KUKA KRL program: UP202.src, UP202.dat

--- UP202.src ---
&ACCESS RV1
&COMMENT WERKZEUGWECHSEL G1
&PARAM EDITMASK = Up999[1-999]
&PARAM TEMPLATE = C:\KRC\Roboter\Template\upvorgabe
&PARAM TPVW_VERSION = 8.3.18
&PARAM DISKPATH = UPs
DEF UP202()
; FOLD UP Anfang;%{SE} %MKUKATPVW
SPS_N=-1
SPS_FERTIG=FALSE
IF NOT CALLBYSELECT THEN
INTERRUPT DECL 10 WHEN $CYCFLAG[254]==FALSE DO VW(#FB_STOP,TRUE)
INTERRUPT ON 10
INT10=TRUE
VW_USR_R (#USR_INIT)
ENDIF
VW(#VW_INIT_UP,TRUE)
; ENDFOLD
;FOLD -- ********************************************** -- ;%{PSE}%MKUKATPVW,%CVW_COM,%VCOMMENT,%P 1:Comment:, 2:**********************************************
;FOLD {H}
M_COMMENT("**********************************************")
;ENDFOLD
;ENDFOLD
;FOLD -- Modell :  VW316/7 -- ;%{PSE}%MKUKATPVW,%CVW_COM,%VCOMMENT,%P 1:Comment:, 2:Modell :  VW316/7
;FOLD {H}
M_COMMENT("Modell :  VW316/7")
;ENDFOLD
;ENDFOLD
;FOLD -- Line   :  TVOL -- ;%{PSE}%MKUKATPVW,%CVW_COM,%VCOMMENT,%P 1:Comment:, 2:Line   :  TVOL
;FOLD {H}
M_COMMENT("Line   :  TVOL")
;ENDFOLD
;ENDFOLD
;FOLD -- Robot  :  5100R01 -- ;%{PSE}%MKUKATPVW,%CVW_COM,%VCOMMENT,%P 1:Comment:, 2:Robot  :  5100R01
;FOLD {H}
M_COMMENT("Robot  :  5100R01")
;ENDFOLD
;ENDFOLD
;FOLD -- Arbeit :  WERKZEUGWECHSEL G2 -- ;%{PSE}%MKUKATPVW,%CVW_COM,%VCOMMENT,%P 1:Comment:, 2:Arbeit :  WERKZEUGWECHSEL G2
;FOLD {H}
M_COMMENT("Arbeit :  WERKZEUGWECHSEL G2")
;ENDFOLD
;ENDFOLD
;FOLD -- ********************************************** -- ;%{PSE}%MKUKATPVW,%CVW_COM,%VCOMMENT,%P 1:Comment:, 2:**********************************************
;FOLD {H}
M_COMMENT("**********************************************")
;ENDFOLD
;ENDFOLD
;FOLD PTP VB=100% VE=0% ACC=100% RobWzg=2 Base=0 SPSTrig=5[1/100s] P;%{P}%MKUKATPVW,%CMOVE8,%VPTP,%P 1:1, 2: VB=, 3:100, 4:%, 5: VE=, 6:0, 7:%, 8: ACC=, 9:100, 10:%, 11: RobWzg=, 12:2, 13: Base=, 14:0, 15: SPSTrig=, 16:5, 17:[1/100s], 18: P, 19:1, 20:-1, 21:1
;FOLD 1:  FB PSPS = EIN;%{SE}%MKUKATPVW %CVW_SPS %VFBPSPS %P 2:FB PSPS = EIN,3:   FBPSPS
;ENDFOLD
;FOLD 2:  -- Initialisierung Merker --;%{SE}%MKUKATPVW %CVW_COM %VCOMMENT %P 2: -- Initialisierung Merker --,3:  VW_COMMENT
;ENDFOLD
;FOLD 3:  SPSMAKRO50 = EIN;%{SE}%MKUKATPVW %CVW_SPS %VMAKRO %P 2:SPSMAKRO50 = EIN,3:   MAKRO
;ENDFOLD
;FOLD 4:  SPSMAKRO51 = EIN;%{SE}%MKUKATPVW %CVW_SPS %VMAKRO %P 2:SPSMAKRO51 = EIN,3:   MAKRO
;ENDFOLD
;FOLD 5:  -- Profilfrei --;%{SE}%MKUKATPVW %CVW_COM %VCOMMENT %P 2: -- Profilfrei --,3:  VW_COMMENT
;ENDFOLD
;FOLD 6:  SPSMAKRO46 = EIN;%{SE}%MKUKATPVW %CVW_SPS %VMAKRO %P 2:SPSMAKRO46 = EIN,3:   MAKRO
;ENDFOLD
;FOLD 7:  -- Verriegelungen Freigabe --;%{SE}%MKUKATPVW %CVW_COM %VCOMMENT %P 2: -- Verriegelungen Freigabe --,3:  VW_COMMENT
;ENDFOLD
;FOLD 8:  SPSMAKRO45 = EIN;%{SE}%MKUKATPVW %CVW_SPS %VMAKRO %P 2:SPSMAKRO45 = EIN,3:   MAKRO
;ENDFOLD
;FOLD 9:  -- Greifer Initialisieren --;%{SE}%MKUKATPVW %CVW_COM %VCOMMENT %P 2: -- Greifer Initialisieren --,3:  VW_COMMENT
;ENDFOLD
;FOLD 10:  F1 = EIN;%{SE}%MKUKATPVW %CVW_SPS %VBOASG %P 2:F1 = EIN,3:   BOASG
;ENDFOLD
;FOLD 11:  F2 = EIN;%{SE}%MKUKATPVW %CVW_SPS %VBOASG %P 2:F2 = EIN,3:   BOASG
;ENDFOLD
;FOLD 12:  F3 = EIN;%{SE}%MKUKATPVW %CVW_SPS %VBOASG %P 2:F3 = EIN,3:   BOASG
;ENDFOLD
;FOLD 13:  F17 = EIN;%{SE}%MKUKATPVW %CVW_SPS %VBOASG %P 2:F17 = EIN,3:   BOASG
;ENDFOLD
;FOLD 14:  M190 = E605 + E603;%{SE}%MKUKATPVW %CVW_SPS %VBOASG %P 2:M190 = E605 + E603,3:   BOASG
;ENDFOLD
;FOLD 15:  SPSMAKRO342 = EIN;%{SE}%MKUKATPVW %CVW_SPS %VMAKRO %P 2:SPSMAKRO342 = EIN,3:   MAKRO
;ENDFOLD
;FOLD 16:  SPSMAKRO340 = EIN;%{SE}%MKUKATPVW %CVW_SPS %VMAKRO %P 2:SPSMAKRO340 = EIN,3:   MAKRO
;ENDFOLD
;FOLD 17:  WARTE BIS M31 & M33 & M35 & M1;%{SE}%MKUKATPVW %CVW_SPS %VWBOASG %P 2:WARTE BIS M31 & M33 & M35 & M1,3:   WBOASG
;ENDFOLD
;FOLD 18:  WARTE BIS E23;%{SE}%MKUKATPVW %CVW_SPS %VWBOASG %P 2:WARTE BIS E23,3:   WBOASG
;ENDFOLD
;FOLD 19:  FB PSPS = M30 & M1 & M31 & M33 & M35;%{SE}%MKUKATPVW %CVW_SPS %VFBPSPS %P 2:FB PSPS = M30 & M1 & M31 & M33 & M35,3:   FBPSPS
;ENDFOLD
;FOLD {H}
VW_MPARA_ACT=P1_D
Act_P1 = P1
Act_P2 = P1
VW(#MPARA,TRUE)
SPS_FERTIG=FALSE
TRIGGER WHEN DISTANCE=1 DELAY=-50 DO SPS_TRIG(1) PRIO=-1
PTP P1
$ADVANCE=1
WAIT FOR SPS_FERTIG
;ENDFOLD
;ENDFOLD
;FOLD -- Werkzeugwechselposition -- ;%{PSE}%MKUKATPVW,%CVW_COM,%VCOMMENT,%P 1:Comment:, 2:Werkzeugwechselposition
;FOLD {H}
M_COMMENT("Werkzeugwechselposition")
;ENDFOLD
;ENDFOLD
;FOLD PTP VB=100% VE=0% ACC=100% RobWzg=2 Base=0 SPSTrig=5[1/100s] P;%{P}%MKUKATPVW,%CMOVE8,%VPTP,%P 1:1, 2: VB=, 3:100, 4:%, 5: VE=, 6:0, 7:%, 8: ACC=, 9:100, 10:%, 11: RobWzg=, 12:2, 13: Base=, 14:0, 15: SPSTrig=, 16:5, 17:[1/100s], 18: P, 19:2, 20:-1, 21:2
;FOLD 1:  FB PSPS = EIN;%{SE}%MKUKATPVW %CVW_SPS %VFBPSPS %P 2:FB PSPS = EIN,3:   FBPSPS
;ENDFOLD
;FOLD 2:  -- Roboter ist in Wartungsstellung --;%{SE}%MKUKATPVW %CVW_COM %VCOMMENT %P 2: -- Roboter ist in Wartungsstellung --,3:  VW_COMMENT
;ENDFOLD
;FOLD 3:  A17 = EIN;%{SE}%MKUKATPVW %CVW_SPS %VBOASG %P 2:A17 = EIN,3:   BOASG
;ENDFOLD
;FOLD 4:  -- Prozessgeraet BMS --;%{SE}%MKUKATPVW %CVW_COM %VCOMMENT %P 2: -- Prozessgeraet BMS --,3:  VW_COMMENT
;ENDFOLD
;FOLD 5:  TECH4 Prozessgeraet  Handling    Greifer=Nr2  in Wartungsstellung   Techaufruf= EIN ;%{SE}%MKUKATPVW %CVW_SPS %VUSER %P 2:    TECH4.Prozessgeraet CN=403 P1=1 P2=0 P3=12 P4=20 P5=0 P6=0 P7=0 P8=0 P9=0 P10=EIN,3:   USER
;ENDFOLD
;FOLD 6:  -- Warte Wartungsstellung Ende --;%{SE}%MKUKATPVW %CVW_COM %VCOMMENT %P 2: -- Warte Wartungsstellung Ende --,3:  VW_COMMENT
;ENDFOLD
;FOLD 7:  WARTE BIS E17;%{SE}%MKUKATPVW %CVW_SPS %VWBOASG %P 2:WARTE BIS E17,3:   WBOASG
;ENDFOLD
;FOLD 8:  -- Wartungsstellung Ende --;%{SE}%MKUKATPVW %CVW_COM %VCOMMENT %P 2: -- Wartungsstellung Ende --,3:  VW_COMMENT
;ENDFOLD
;FOLD 9:  A17 = AUS;%{SE}%MKUKATPVW %CVW_SPS %VBOASG %P 2:A17 = AUS,3:   BOASG
;ENDFOLD
;FOLD 10:  WARTE BIS E23;%{SE}%MKUKATPVW %CVW_SPS %VWBOASG %P 2:WARTE BIS E23,3:   WBOASG
;ENDFOLD
;FOLD 11:  FB PSPS = M30 & M1 & M31 & M33 & M35;%{SE}%MKUKATPVW %CVW_SPS %VFBPSPS %P 2:FB PSPS = M30 & M1 & M31 & M33 & M35,3:   FBPSPS
;ENDFOLD
;FOLD {H}
VW_MPARA_ACT=P2_D
Act_P1 = P2
Act_P2 = P2
VW(#MPARA,TRUE)
SPS_FERTIG=FALSE
TRIGGER WHEN DISTANCE=1 DELAY=-50 DO SPS_TRIG(2) PRIO=-1
VW_USER (#USR_ADV,403,1,0,12,20,0,0,0,0,0,TRUE)
VW_USR_R (#USR_ADV,403,1,0,12,20,0,0,0,0,0,TRUE)
PTP P2
$ADVANCE=1
WAIT FOR SPS_FERTIG
VW_USER (#USR_MAIN,403,1,0,12,20,0,0,0,0,0,TRUE)
VW_USR_R (#USR_MAIN,403,1,0,12,20,0,0,0,0,0,TRUE)
;ENDFOLD
;ENDFOLD
;FOLD PTP VB=100% VE=0% ACC=100% RobWzg=2 Base=0 SPSTrig=5[1/100s] P;%{P}%MKUKATPVW,%CMOVE8,%VPTP,%P 1:1, 2: VB=, 3:100, 4:%, 5: VE=, 6:0, 7:%, 8: ACC=, 9:100, 10:%, 11: RobWzg=, 12:2, 13: Base=, 14:0, 15: SPSTrig=, 16:5, 17:[1/100s], 18: P, 19:3, 20:-1, 21:3
;FOLD 1:  FB PSPS = EIN;%{SE}%MKUKATPVW %CVW_SPS %VFBPSPS %P 2:FB PSPS = EIN,3:   FBPSPS
;ENDFOLD
;FOLD 2:  WARTE BIS E23;%{SE}%MKUKATPVW %CVW_SPS %VWBOASG %P 2:WARTE BIS E23,3:   WBOASG
;ENDFOLD
;FOLD 3:  FB PSPS = M30 & M1 & M31 & M33 & M35;%{SE}%MKUKATPVW %CVW_SPS %VFBPSPS %P 2:FB PSPS = M30 & M1 & M31 & M33 & M35,3:   FBPSPS
;ENDFOLD
;FOLD {H}
VW_MPARA_ACT=P3_D
Act_P1 = P3
Act_P2 = P3
VW(#MPARA,TRUE)
SPS_FERTIG=FALSE
TRIGGER WHEN DISTANCE=1 DELAY=-50 DO SPS_TRIG(3) PRIO=-1
PTP P3
$ADVANCE=1
WAIT FOR SPS_FERTIG
;ENDFOLD
;ENDFOLD
; FOLD ;%{H}
END
DEF SPS_TRIG(NO :IN)
INT NO
INT VW_STOP
BOOL UES
BOOL ANA_UES
BOOL ANA_TRIG
VW_STOP=$VW_PSPS_STOP
UES=FALSE
ANA_UES=FALSE
ANA_TRIG=FALSE
IF ((NO>10000) AND (NO<20000)) THEN
NO=NO-10000
UES=TRUE
ENDIF
IF ((NO>20000) AND (NO<30000)) THEN
NO=NO-20000
ANA_TRIG=TRUE
ENDIF
IF NO>30000 THEN
NO=NO-30000
ANA_UES=TRUE
ANA_TRIG=TRUE
ENDIF
; FOLD ;%{H}
IF ((VW_STOP B_AND 'B0001') > 0) THEN
;-- Trigger vorzeitig geschaltet (delay < 0) oder MStep
IF (((VW_STOP B_AND 'B0110') > 0) AND ($MODE_OP<>#EX)) THEN
;-- MStep oder BCO Bewegung
HALT
ENDIF
ENDIF
; ENDFOLD
IF (SEARCH_END) THEN
SEARCH_END = FALSE
INTERRUPT OFF 39
ENDIF
SWITCH NO
CASE 1
;FOLD SPS_TRIG1 {H}
VALCYCFL30=$CYCFLAG[254]
$CYCFLAG[254]=(TRUE) AND $CYCFLAG[255] OR ($TIMER[61]<0)
VW(#FB_CHECK,TRUE)
SEL_RES = SELECT (#MAKRO,50,TRUE,,,,,FALSE)
SEL_RES = SELECT (#MAKRO,51,TRUE,,,,,FALSE)
SEL_RES = SELECT (#MAKRO,46,TRUE,,,,,FALSE)
SEL_RES = SELECT (#MAKRO,45,TRUE,,,,,FALSE)
$FLAG[1]=TRUE
$FLAG[2]=TRUE
$FLAG[3]=TRUE
$FLAG[17]=TRUE
$CYCFLAG[190]=$IN[605] OR $IN[603]
SEL_RES = SELECT (#MAKRO,342,TRUE,,,,,FALSE)
SEL_RES = SELECT (#MAKRO,340,TRUE,,,,,FALSE)
$LOOP_MSG[]="M31 & M33 & M35 & M1"
$LOOP_CONT=TRUE
WAIT FOR ($CYCFLAG[31] AND $CYCFLAG[33] AND $CYCFLAG[35] AND $CYCFLAG[1]) OR (NOT $LOOP_CONT AND ($MODE_OP<>#EX))
$LOOP_MSG[]="                                                                                                                                "
$LOOP_MSG[]="E23"
$LOOP_CONT=TRUE
WAIT FOR ($IN[23]) OR (NOT $LOOP_CONT AND ($MODE_OP<>#EX))
$LOOP_MSG[]="                                                                                                                                "
VALCYCFL30=$CYCFLAG[254]
$CYCFLAG[254]=($CYCFLAG[30] AND $CYCFLAG[1] AND $CYCFLAG[31] AND $CYCFLAG[33] AND $CYCFLAG[35]) AND $CYCFLAG[255] OR ($TIMER[61]<0)
VW(#FB_CHECK,TRUE)
;ENDFOLD
CASE 2
;FOLD SPS_TRIG2 {H}
VALCYCFL30=$CYCFLAG[254]
$CYCFLAG[254]=(TRUE) AND $CYCFLAG[255] OR ($TIMER[61]<0)
VW(#FB_CHECK,TRUE)
$OUT[17]=TRUE
VW_USER (#USR_TRIG,403,1,0,12,20,0,0,0,0,0,TRUE)
VW_USR_R (#USR_TRIG,403,1,0,12,20,0,0,0,0,0,TRUE)
$LOOP_MSG[]="E17"
$LOOP_CONT=TRUE
WAIT FOR ($IN[17]) OR (NOT $LOOP_CONT AND ($MODE_OP<>#EX))
$LOOP_MSG[]="                                                                                                                                "
$OUT[17]=FALSE
$LOOP_MSG[]="E23"
$LOOP_CONT=TRUE
WAIT FOR ($IN[23]) OR (NOT $LOOP_CONT AND ($MODE_OP<>#EX))
$LOOP_MSG[]="                                                                                                                                "
VALCYCFL30=$CYCFLAG[254]
$CYCFLAG[254]=($CYCFLAG[30] AND $CYCFLAG[1] AND $CYCFLAG[31] AND $CYCFLAG[33] AND $CYCFLAG[35]) AND $CYCFLAG[255] OR ($TIMER[61]<0)
VW(#FB_CHECK,TRUE)
;ENDFOLD
CASE 3
;FOLD SPS_TRIG3 {H}
VALCYCFL30=$CYCFLAG[254]
$CYCFLAG[254]=(TRUE) AND $CYCFLAG[255] OR ($TIMER[61]<0)
VW(#FB_CHECK,TRUE)
$LOOP_MSG[]="E23"
$LOOP_CONT=TRUE
WAIT FOR ($IN[23]) OR (NOT $LOOP_CONT AND ($MODE_OP<>#EX))
$LOOP_MSG[]="                                                                                                                                "
VALCYCFL30=$CYCFLAG[254]
$CYCFLAG[254]=($CYCFLAG[30] AND $CYCFLAG[1] AND $CYCFLAG[31] AND $CYCFLAG[33] AND $CYCFLAG[35]) AND $CYCFLAG[255] OR ($TIMER[61]<0)
VW(#FB_CHECK,TRUE)
;ENDFOLD
CASE 4
;FOLD SPS_TRIG4 {H}
;ENDFOLD
CASE 5
;FOLD SPS_TRIG5 {H}
;ENDFOLD
CASE 6
;FOLD SPS_TRIG6 {H}
;ENDFOLD
CASE 7
;FOLD SPS_TRIG7 {H}
;ENDFOLD
CASE 8
;FOLD SPS_TRIG8 {H}
;ENDFOLD
CASE 9
;FOLD SPS_TRIG9 {H}
;ENDFOLD
CASE 10
;FOLD SPS_TRIG10 {H}
;ENDFOLD
CASE 11
;FOLD SPS_TRIG11 {H}
;ENDFOLD
CASE 12
;FOLD SPS_TRIG12 {H}
;ENDFOLD
CASE 13
;FOLD SPS_TRIG13 {H}
;ENDFOLD
CASE 14
;FOLD SPS_TRIG14 {H}
;ENDFOLD
CASE 15
;FOLD SPS_TRIG15 {H}
;ENDFOLD
CASE 16
;FOLD SPS_TRIG16 {H}
;ENDFOLD
CASE 17
;FOLD SPS_TRIG17 {H}
;ENDFOLD
CASE 18
;FOLD SPS_TRIG18 {H}
;ENDFOLD
CASE 19
;FOLD SPS_TRIG19 {H}
;ENDFOLD
CASE 20
;FOLD SPS_TRIG20 {H}
;ENDFOLD
CASE 21
;FOLD SPS_TRIG21 {H}
;ENDFOLD
CASE 22
;FOLD SPS_TRIG22 {H}
;ENDFOLD
CASE 23
;FOLD SPS_TRIG23 {H}
;ENDFOLD
CASE 24
;FOLD SPS_TRIG24 {H}
;ENDFOLD
CASE 25
;FOLD SPS_TRIG25 {H}
;ENDFOLD
CASE 26
;FOLD SPS_TRIG26 {H}
;ENDFOLD
CASE 27
;FOLD SPS_TRIG27 {H}
;ENDFOLD
CASE 28
;FOLD SPS_TRIG28 {H}
;ENDFOLD
CASE 29
;FOLD SPS_TRIG29 {H}
;ENDFOLD
CASE 30
;FOLD SPS_TRIG30 {H}
;ENDFOLD
CASE 31
;FOLD SPS_TRIG31 {H}
;ENDFOLD
CASE 32
;FOLD SPS_TRIG32 {H}
;ENDFOLD
CASE 33
;FOLD SPS_TRIG33 {H}
;ENDFOLD
CASE 34
;FOLD SPS_TRIG34 {H}
;ENDFOLD
CASE 35
;FOLD SPS_TRIG35 {H}
;ENDFOLD
CASE 36
;FOLD SPS_TRIG36 {H}
;ENDFOLD
CASE 37
;FOLD SPS_TRIG37 {H}
;ENDFOLD
CASE 38
;FOLD SPS_TRIG38 {H}
;ENDFOLD
CASE 39
;FOLD SPS_TRIG39 {H}
;ENDFOLD
CASE 40
;FOLD SPS_TRIG40 {H}
;ENDFOLD
CASE 41
;FOLD SPS_TRIG41 {H}
;ENDFOLD
CASE 42
;FOLD SPS_TRIG42 {H}
;ENDFOLD
CASE 43
;FOLD SPS_TRIG43 {H}
;ENDFOLD
CASE 44
;FOLD SPS_TRIG44 {H}
;ENDFOLD
CASE 45
;FOLD SPS_TRIG45 {H}
;ENDFOLD
CASE 46
;FOLD SPS_TRIG46 {H}
;ENDFOLD
CASE 47
;FOLD SPS_TRIG47 {H}
;ENDFOLD
CASE 48
;FOLD SPS_TRIG48 {H}
;ENDFOLD
CASE 49
;FOLD SPS_TRIG49 {H}
;ENDFOLD
CASE 50
;FOLD SPS_TRIG50 {H}
;ENDFOLD
CASE 51
;FOLD SPS_TRIG51 {H}
;ENDFOLD
CASE 52
;FOLD SPS_TRIG52 {H}
;ENDFOLD
CASE 53
;FOLD SPS_TRIG53 {H}
;ENDFOLD
CASE 54
;FOLD SPS_TRIG54 {H}
;ENDFOLD
CASE 55
;FOLD SPS_TRIG55 {H}
;ENDFOLD
CASE 56
;FOLD SPS_TRIG56 {H}
;ENDFOLD
CASE 57
;FOLD SPS_TRIG57 {H}
;ENDFOLD
CASE 58
;FOLD SPS_TRIG58 {H}
;ENDFOLD
CASE 59
;FOLD SPS_TRIG59 {H}
;ENDFOLD
CASE 60
;FOLD SPS_TRIG60 {H}
;ENDFOLD
CASE 61
;FOLD SPS_TRIG61 {H}
;ENDFOLD
CASE 62
;FOLD SPS_TRIG62 {H}
;ENDFOLD
CASE 63
;FOLD SPS_TRIG63 {H}
;ENDFOLD
CASE 64
;FOLD SPS_TRIG64 {H}
;ENDFOLD
CASE 65
;FOLD SPS_TRIG65 {H}
;ENDFOLD
CASE 66
;FOLD SPS_TRIG66 {H}
;ENDFOLD
CASE 67
;FOLD SPS_TRIG67 {H}
;ENDFOLD
CASE 68
;FOLD SPS_TRIG68 {H}
;ENDFOLD
CASE 69
;FOLD SPS_TRIG69 {H}
;ENDFOLD
CASE 70
;FOLD SPS_TRIG70 {H}
;ENDFOLD
CASE 71
;FOLD SPS_TRIG71 {H}
;ENDFOLD
CASE 72
;FOLD SPS_TRIG72 {H}
;ENDFOLD
CASE 73
;FOLD SPS_TRIG73 {H}
;ENDFOLD
CASE 74
;FOLD SPS_TRIG74 {H}
;ENDFOLD
CASE 75
;FOLD SPS_TRIG75 {H}
;ENDFOLD
CASE 76
;FOLD SPS_TRIG76 {H}
;ENDFOLD
CASE 77
;FOLD SPS_TRIG77 {H}
;ENDFOLD
CASE 78
;FOLD SPS_TRIG78 {H}
;ENDFOLD
CASE 79
;FOLD SPS_TRIG79 {H}
;ENDFOLD
CASE 80
;FOLD SPS_TRIG80 {H}
;ENDFOLD
CASE 81
;FOLD SPS_TRIG81 {H}
;ENDFOLD
CASE 82
;FOLD SPS_TRIG82 {H}
;ENDFOLD
CASE 83
;FOLD SPS_TRIG83 {H}
;ENDFOLD
CASE 84
;FOLD SPS_TRIG84 {H}
;ENDFOLD
CASE 85
;FOLD SPS_TRIG85 {H}
;ENDFOLD
CASE 86
;FOLD SPS_TRIG86 {H}
;ENDFOLD
CASE 87
;FOLD SPS_TRIG87 {H}
;ENDFOLD
CASE 88
;FOLD SPS_TRIG88 {H}
;ENDFOLD
CASE 89
;FOLD SPS_TRIG89 {H}
;ENDFOLD
CASE 90
;FOLD SPS_TRIG90 {H}
;ENDFOLD
CASE 91
;FOLD SPS_TRIG91 {H}
;ENDFOLD
CASE 92
;FOLD SPS_TRIG92 {H}
;ENDFOLD
CASE 93
;FOLD SPS_TRIG93 {H}
;ENDFOLD
CASE 94
;FOLD SPS_TRIG94 {H}
;ENDFOLD
CASE 95
;FOLD SPS_TRIG95 {H}
;ENDFOLD
CASE 96
;FOLD SPS_TRIG96 {H}
;ENDFOLD
CASE 97
;FOLD SPS_TRIG97 {H}
;ENDFOLD
CASE 98
;FOLD SPS_TRIG98 {H}
;ENDFOLD
CASE 99
;FOLD SPS_TRIG99 {H}
;ENDFOLD
CASE 100
;FOLD SPS_TRIG100 {H}
;ENDFOLD
CASE 101
;FOLD SPS_TRIG101 {H}
;ENDFOLD
CASE 102
;FOLD SPS_TRIG102 {H}
;ENDFOLD
CASE 103
;FOLD SPS_TRIG103 {H}
;ENDFOLD
CASE 104
;FOLD SPS_TRIG104 {H}
;ENDFOLD
CASE 105
;FOLD SPS_TRIG105 {H}
;ENDFOLD
CASE 106
;FOLD SPS_TRIG106 {H}
;ENDFOLD
CASE 107
;FOLD SPS_TRIG107 {H}
;ENDFOLD
CASE 108
;FOLD SPS_TRIG108 {H}
;ENDFOLD
CASE 109
;FOLD SPS_TRIG109 {H}
;ENDFOLD
CASE 110
;FOLD SPS_TRIG110 {H}
;ENDFOLD
CASE 111
;FOLD SPS_TRIG111 {H}
;ENDFOLD
CASE 112
;FOLD SPS_TRIG112 {H}
;ENDFOLD
CASE 113
;FOLD SPS_TRIG113 {H}
;ENDFOLD
CASE 114
;FOLD SPS_TRIG114 {H}
;ENDFOLD
CASE 115
;FOLD SPS_TRIG115 {H}
;ENDFOLD
CASE 116
;FOLD SPS_TRIG116 {H}
;ENDFOLD
CASE 117
;FOLD SPS_TRIG117 {H}
;ENDFOLD
CASE 118
;FOLD SPS_TRIG118 {H}
;ENDFOLD
CASE 119
;FOLD SPS_TRIG119 {H}
;ENDFOLD
CASE 120
;FOLD SPS_TRIG120 {H}
;ENDFOLD
CASE 121
;FOLD SPS_TRIG121 {H}
;ENDFOLD
CASE 122
;FOLD SPS_TRIG122 {H}
;ENDFOLD
CASE 123
;FOLD SPS_TRIG123 {H}
;ENDFOLD
CASE 124
;FOLD SPS_TRIG124 {H}
;ENDFOLD
CASE 125
;FOLD SPS_TRIG125 {H}
;ENDFOLD
CASE 126
;FOLD SPS_TRIG126 {H}
;ENDFOLD
CASE 127
;FOLD SPS_TRIG127 {H}
;ENDFOLD
CASE 128
;FOLD SPS_TRIG128 {H}
;ENDFOLD
CASE 129
;FOLD SPS_TRIG129 {H}
;ENDFOLD
CASE 130
;FOLD SPS_TRIG130 {H}
;ENDFOLD
CASE 131
;FOLD SPS_TRIG131 {H}
;ENDFOLD
CASE 132
;FOLD SPS_TRIG132 {H}
;ENDFOLD
CASE 133
;FOLD SPS_TRIG133 {H}
;ENDFOLD
CASE 134
;FOLD SPS_TRIG134 {H}
;ENDFOLD
CASE 135
;FOLD SPS_TRIG135 {H}
;ENDFOLD
CASE 136
;FOLD SPS_TRIG136 {H}
;ENDFOLD
CASE 137
;FOLD SPS_TRIG137 {H}
;ENDFOLD
CASE 138
;FOLD SPS_TRIG138 {H}
;ENDFOLD
CASE 139
;FOLD SPS_TRIG139 {H}
;ENDFOLD
CASE 140
;FOLD SPS_TRIG140 {H}
;ENDFOLD
CASE 141
;FOLD SPS_TRIG141 {H}
;ENDFOLD
CASE 142
;FOLD SPS_TRIG142 {H}
;ENDFOLD
CASE 143
;FOLD SPS_TRIG143 {H}
;ENDFOLD
CASE 144
;FOLD SPS_TRIG144 {H}
;ENDFOLD
CASE 145
;FOLD SPS_TRIG145 {H}
;ENDFOLD
CASE 146
;FOLD SPS_TRIG146 {H}
;ENDFOLD
CASE 147
;FOLD SPS_TRIG147 {H}
;ENDFOLD
CASE 148
;FOLD SPS_TRIG148 {H}
;ENDFOLD
CASE 149
;FOLD SPS_TRIG149 {H}
;ENDFOLD
CASE 150
;FOLD SPS_TRIG150 {H}
;ENDFOLD
CASE 151
;FOLD SPS_TRIG151 {H}
;ENDFOLD
CASE 152
;FOLD SPS_TRIG152 {H}
;ENDFOLD
CASE 153
;FOLD SPS_TRIG153 {H}
;ENDFOLD
CASE 154
;FOLD SPS_TRIG154 {H}
;ENDFOLD
CASE 155
;FOLD SPS_TRIG155 {H}
;ENDFOLD
CASE 156
;FOLD SPS_TRIG156 {H}
;ENDFOLD
CASE 157
;FOLD SPS_TRIG157 {H}
;ENDFOLD
CASE 158
;FOLD SPS_TRIG158 {H}
;ENDFOLD
CASE 159
;FOLD SPS_TRIG159 {H}
;ENDFOLD
CASE 160
;FOLD SPS_TRIG160 {H}
;ENDFOLD
CASE 161
;FOLD SPS_TRIG161 {H}
;ENDFOLD
CASE 162
;FOLD SPS_TRIG162 {H}
;ENDFOLD
CASE 163
;FOLD SPS_TRIG163 {H}
;ENDFOLD
CASE 164
;FOLD SPS_TRIG164 {H}
;ENDFOLD
CASE 165
;FOLD SPS_TRIG165 {H}
;ENDFOLD
CASE 166
;FOLD SPS_TRIG166 {H}
;ENDFOLD
CASE 167
;FOLD SPS_TRIG167 {H}
;ENDFOLD
CASE 168
;FOLD SPS_TRIG168 {H}
;ENDFOLD
CASE 169
;FOLD SPS_TRIG169 {H}
;ENDFOLD
CASE 170
;FOLD SPS_TRIG170 {H}
;ENDFOLD
CASE 171
;FOLD SPS_TRIG171 {H}
;ENDFOLD
CASE 172
;FOLD SPS_TRIG172 {H}
;ENDFOLD
CASE 173
;FOLD SPS_TRIG173 {H}
;ENDFOLD
CASE 174
;FOLD SPS_TRIG174 {H}
;ENDFOLD
CASE 175
;FOLD SPS_TRIG175 {H}
;ENDFOLD
CASE 176
;FOLD SPS_TRIG176 {H}
;ENDFOLD
CASE 177
;FOLD SPS_TRIG177 {H}
;ENDFOLD
CASE 178
;FOLD SPS_TRIG178 {H}
;ENDFOLD
CASE 179
;FOLD SPS_TRIG179 {H}
;ENDFOLD
CASE 180
;FOLD SPS_TRIG180 {H}
;ENDFOLD
CASE 181
;FOLD SPS_TRIG181 {H}
;ENDFOLD
CASE 182
;FOLD SPS_TRIG182 {H}
;ENDFOLD
CASE 183
;FOLD SPS_TRIG183 {H}
;ENDFOLD
CASE 184
;FOLD SPS_TRIG184 {H}
;ENDFOLD
CASE 185
;FOLD SPS_TRIG185 {H}
;ENDFOLD
CASE 186
;FOLD SPS_TRIG186 {H}
;ENDFOLD
CASE 187
;FOLD SPS_TRIG187 {H}
;ENDFOLD
CASE 188
;FOLD SPS_TRIG188 {H}
;ENDFOLD
CASE 189
;FOLD SPS_TRIG189 {H}
;ENDFOLD
CASE 190
;FOLD SPS_TRIG190 {H}
;ENDFOLD
CASE 191
;FOLD SPS_TRIG191 {H}
;ENDFOLD
CASE 192
;FOLD SPS_TRIG192 {H}
;ENDFOLD
CASE 193
;FOLD SPS_TRIG193 {H}
;ENDFOLD
CASE 194
;FOLD SPS_TRIG194 {H}
;ENDFOLD
CASE 195
;FOLD SPS_TRIG195 {H}
;ENDFOLD
CASE 196
;FOLD SPS_TRIG196 {H}
;ENDFOLD
CASE 197
;FOLD SPS_TRIG197 {H}
;ENDFOLD
CASE 198
;FOLD SPS_TRIG198 {H}
;ENDFOLD
CASE 199
;FOLD SPS_TRIG199 {H}
;ENDFOLD
CASE 200
;FOLD SPS_TRIG200 {H}
;ENDFOLD
CASE 201
;FOLD SPS_TRIG201 {H}
;ENDFOLD
CASE 202
;FOLD SPS_TRIG202 {H}
;ENDFOLD
CASE 203
;FOLD SPS_TRIG203 {H}
;ENDFOLD
CASE 204
;FOLD SPS_TRIG204 {H}
;ENDFOLD
CASE 205
;FOLD SPS_TRIG205 {H}
;ENDFOLD
CASE 206
;FOLD SPS_TRIG206 {H}
;ENDFOLD
CASE 207
;FOLD SPS_TRIG207 {H}
;ENDFOLD
CASE 208
;FOLD SPS_TRIG208 {H}
;ENDFOLD
CASE 209
;FOLD SPS_TRIG209 {H}
;ENDFOLD
CASE 210
;FOLD SPS_TRIG210 {H}
;ENDFOLD
CASE 211
;FOLD SPS_TRIG211 {H}
;ENDFOLD
DEFAULT
ENDSWITCH
; FOLD ;%{H}
IF ($MODE_OP<>#EX) THEN
;-- Trigger erst nach Wiederanstart geschaltet --
IF ((((VW_STOP B_AND 'B10010') >0) AND ((VW_STOP B_AND 'B0001')<=0))) THEN
;-- MStep Bewegung --
HALT
ENDIF
ENDIF
; ENDFOLD
IF (NOT UES AND NOT ANA_TRIG) THEN
SPS_FERTIG=TRUE
ENDIF
IF (NOT ANA_UES AND ANA_TRIG) THEN
SPS_FERTIG_ANA=TRUE
ENDIF
END
; ENDFOLD

--- UP202.dat ---
&ACCESS RV1
&COMMENT WERKZEUGWECHSEL G1
&PARAM EDITMASK = Up999[1-999]
&PARAM TEMPLATE = C:\KRC\Roboter\Template\upvorgabe
&PARAM TPVW_VERSION = 8.3.18
&PARAM DISKPATH = UPs
DEFDAT  UP202
; FOLD ;%{H} %MKUKATPVW
; ENDFOLD
; interface to basic routines
EXT  BAS (BAS_COMMAND  :IN,REAL  :IN )
; interface to VW-standard routines
EXT  VW (VW_COMMAND  :IN,BOOL  :IN,REAL  :IN,REAL  :IN,REAL  :IN,REAL  :IN,BOOL  :IN,E6POS  :IN )
; interface to VW_USER - Call
EXT  VW_USER (VW_USER_CMD  :IN,INT  :IN,REAL  :IN,REAL  :IN,REAL  :IN,REAL  :IN,REAL  :IN,REAL  :IN,REAL  :IN,REAL  :IN,REAL  :IN,BOOL  :IN )
EXT  VW_USR_R (VW_USER_CMD  :IN,INT  :IN,REAL  :IN,REAL  :IN,REAL  :IN,REAL  :IN,REAL  :IN,REAL  :IN,REAL  :IN,REAL  :IN,REAL  :IN,BOOL  :IN )
EXT  IBGN (IBGN_COMMAND  :IN,BOOL  :IN,REAL  :IN,REAL  :IN,BOOL  :IN,E6POS  :OUT )
; interface select routine
EXTFCT  INT  SELECT(SUBTYPE  :IN,INT  :IN,BOOL  :IN,ARI_TYP  :IN,INT  :IN,BOOL_TYP  :IN,INT  :IN,BOOL  :IN)
INT VW_NEXT_FREE=4
INT VW_NFREE_SPS=4
INT VW_MAX_SPS=211
DECL VW_MPARA_TYP P1_D={TOOL_NO 2,BASE_NO 0,VB 100,VE 0,ACC 100,TRG_TIME 5,MOVE_TYPE #PTP_MOTION}
DECL E6POS P1={X 273.551483,Y 1212.98267,Z 954.982666,A -175.620789,B 82.2778244,C -49.8938828,S 2,T 3,E1 -518.843384,E2 0.0,E3 0.0,E4 0.0,E5 0.0,E6 0.0}
DECL VW_MPARA_TYP P2_D={TOOL_NO 2,BASE_NO 0,VB 100,VE 0,ACC 100,TRG_TIME 5,MOVE_TYPE #PTP_MOTION}
DECL E6POS P2={X 273.551483,Y 1212.98267,Z 954.982666,A -175.620789,B 82.2778244,C -49.8938828,S 2,T 3,E1 -518.843384,E2 0.0,E3 0.0,E4 0.0,E5 0.0,E6 0.0}
DECL VW_MPARA_TYP P3_D={TOOL_NO 2,BASE_NO 0,VB 100,VE 0,ACC 100,TRG_TIME 5,MOVE_TYPE #PTP_MOTION}
DECL E6POS P3={X 273.551483,Y 1212.98267,Z 954.982666,A -175.620789,B 82.2778244,C -49.8938828,S 2,T 3,E1 -518.843384,E2 0.0,E3 0.0,E4 0.0,E5 0.0,E6 0.0}
ENDDAT
